FUNCTION_BLOCK FB_BinaryDevice EXTENDS FB_HMIBase
VAR
	binary : Discrete.I_DiscreteBase;
END_VAR

METHOD Cyclic
VAR
END_VAR
// Sync status from device to HMI
status.HmiStatus.Busy := binary.P_DiscreteStatus.ComponentStatus.BaseStatus.Busy;
status.HmiStatus.Done := binary.P_DiscreteStatus.ComponentStatus.BaseStatus.Done;
status.HmiStatus.Error := binary.P_DiscreteStatus.ComponentStatus.BaseStatus.Error;

// Map discrete state to Enabled flag
status.HmiStatus.Enabled := (binary.P_DiscreteStatus.BinaryComponentState = Discrete.E_DiscreteComponentState.Active);

// Handle commands from Vue.js
IF cmd.Enable THEN
	binary.Activate();
	cmd.Enable := FALSE;
END_IF

IF cmd.Disable THEN
	binary.Deactivate();
	cmd.Disable := FALSE;
END_IF
END_METHOD

METHOD Init : BOOL
VAR_INPUT
	refBinary : Discrete.I_DiscreteBase;
END_VAR
binary := refBinary;
Init := TRUE;
END_METHOD

END_FUNCTION_BLOCK

(* stored: Version 1.1.0.1
   POU FB_BinaryDevice: Id {1f2462be-444f-471b-ae3d-f444ab9627ba}, SpecialFunc None
   Method Cyclic: Id {1c7bbb0e-cba7-43ac-bb5d-4c2b907180fc}
   Method Init: Id {6885a98e-288a-434d-ba1e-96376fb179a6} *)
